Staubli VAL3: onEnterEvent.pgx

program onEnterEvent(bool& x_bSave (dimensions=1))
begin
  //
  // NB sEvent is the selected
  // element in the LIST
  //
  if nIndex==0
    // change the name
    call changePoint(0)
  else
    if (nIndex-nUserItem)>0
      // change the default value
      call changePoint(nIndex-nUserItem)
      x_bSave=true
    else
      // change the custom item
      call trajType:onEditItem(sEvent,nIndex-1,nIndexItem)
    endIf
  endIf
  x_bSave=true
  call buildList()
end
